{attribute addProperty BoxType "AX5203-0000-0005-0005"}
{attribute addProperty Id "AT_xAT %I*ARRAY[0..1] OF AT_029F011596120MDTAT %Q*ARRAY[0..1] OF MDT_47A878CF96120WcStateAT %I*WcState_F855686C1620InfoDataAT %I*InfoData_81099714160200"}
{attribute addProperty CRC "1704960465"}
{attribute addProperty SizeInBites "368"}
{attribute addProperty SizeInBytes "46"}
TYPE AX5203_4DACCC4B :
STRUCT
	{attribute addProperty Name "AT"}
	AT_x : ARRAY[0..1] OF AT_029F0115;
	{attribute addProperty Name "MDT"}
	MDT : ARRAY[0..1] OF MDT_47A878CF;
	{attribute addProperty Name "WcState"}
	WcState : WcState_F855686C;
	{attribute addProperty Name "InfoData"}
	InfoData : InfoData_81099714;
END_STRUCT
END_TYPE

(* stored: Version 1.2.0.0, ProductVersion 3.1.4024.9
   DUT AX5203_4DACCC4B: Id {d8d20ec4-c31f-48b7-bd83-fb1a7a3f5020} *)
